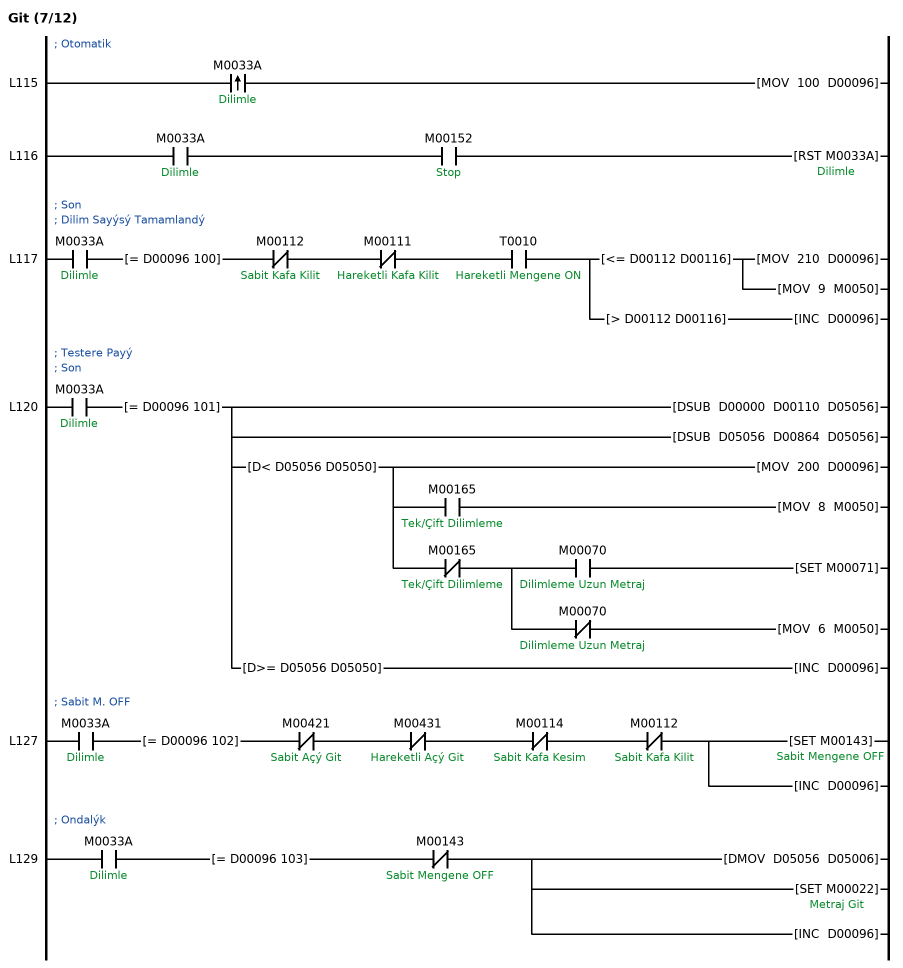
; L115
LOADP     M0033A	// Dilimle
MOV       100 D00096
// output comment: Otomatik
; L116
LOAD      M0033A	// Dilimle
AND       M00152	// Stop
RST       M0033A	// Dilimle
; L117
LOAD      M0033A	// Dilimle
AND=      D00096 100
AND NOT   M00112	// Sabit Kafa Kilit
AND NOT   M00111	// Hareketli Kafa Kilit
AND       T0010	// Hareketli Mengene ON
MPUSH
AND<=     D00112 D00116
MOV       210 D00096
MOV       9 M0050
MPOP
AND>      D00112 D00116
INC       D00096
// output comment: Son
// output comment: Dilim Sayýsý Tamamlandý
; L120
LOAD      M0033A	// Dilimle
AND=      D00096 101
DSUB      D00000 D00110 D05056
DSUB      D05056 D00864 D05056
MPUSH
ANDD<     D05056 D05050
MOV       200 D00096
MPUSH
AND       M00165	// Tek/Çift Dilimleme
MOV       8 M0050
MPOP
AND NOT   M00165	// Tek/Çift Dilimleme
MPUSH
AND       M00070	// Dilimleme Uzun Metraj
SET       M00071
MPOP
AND NOT   M00070	// Dilimleme Uzun Metraj
MOV       6 M0050
MPOP
ANDD>=    D05056 D05050
INC       D00096
// output comment: Testere Payý
// output comment: Son
; L127
LOAD      M0033A	// Dilimle
AND=      D00096 102
AND NOT   M00421	// Sabit Açý Git
AND NOT   M00431	// Hareketli Açý Git
AND NOT   M00114	// Sabit Kafa Kesim
AND NOT   M00112	// Sabit Kafa Kilit
SET       M00143	// Sabit Mengene OFF
INC       D00096
// output comment: Sabit M. OFF
; L129
LOAD      M0033A	// Dilimle
AND=      D00096 103
AND NOT   M00143	// Sabit Mengene OFF
DMOV      D05056 D05006
SET       M00022	// Metraj Git
INC       D00096
// output comment: Ondalýk

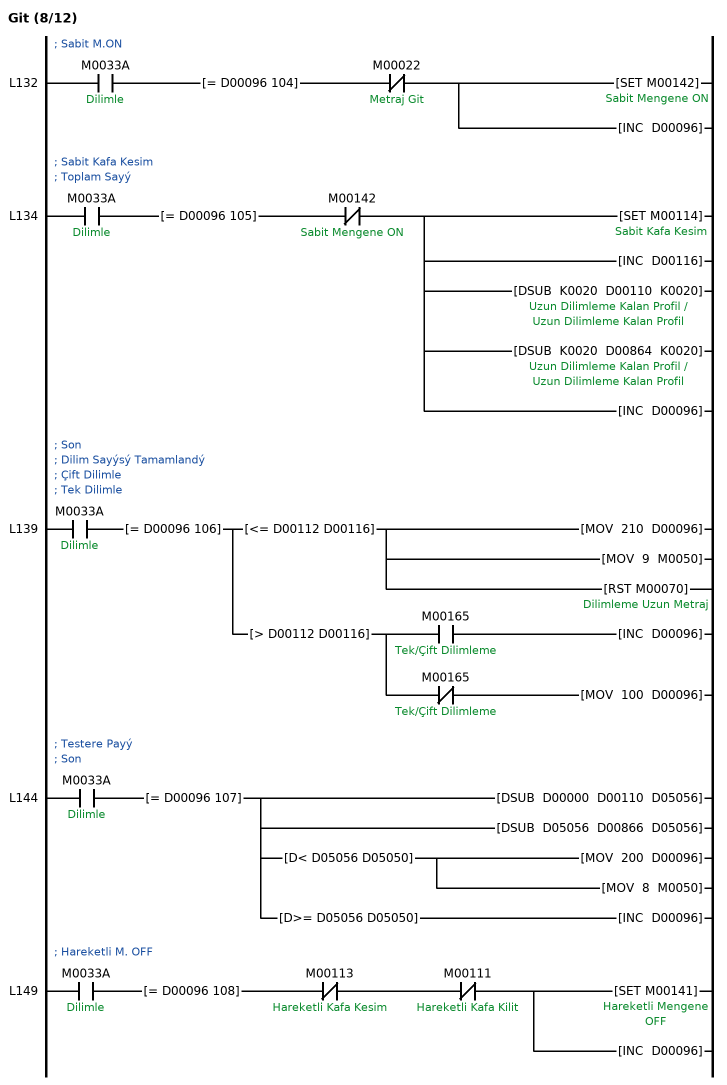
; L132
LOAD      M0033A	// Dilimle
AND=      D00096 104
AND NOT   M00022	// Metraj Git
SET       M00142	// Sabit Mengene ON
INC       D00096
// output comment: Sabit M.ON
; L134
LOAD      M0033A	// Dilimle
AND=      D00096 105
AND NOT   M00142	// Sabit Mengene ON
SET       M00114	// Sabit Kafa Kesim
INC       D00116
DSUB      K0020 D00110 K0020	// Uzun Dilimleme Kalan Profil / Uzun Dilimleme Kalan Profil
DSUB      K0020 D00864 K0020	// Uzun Dilimleme Kalan Profil / Uzun Dilimleme Kalan Profil
INC       D00096
// output comment: Sabit Kafa Kesim
// output comment: Toplam Sayý
; L139
LOAD      M0033A	// Dilimle
AND=      D00096 106
MPUSH
AND<=     D00112 D00116
MOV       210 D00096
MOV       9 M0050
RST       M00070	// Dilimleme Uzun Metraj
MPOP
AND>      D00112 D00116
MPUSH
AND       M00165	// Tek/Çift Dilimleme
INC       D00096
MPOP
AND NOT   M00165	// Tek/Çift Dilimleme
MOV       100 D00096
// output comment: Son
// output comment: Dilim Sayýsý Tamamlandý
// output comment: Çift Dilimle
// output comment: Tek Dilimle
; L144
LOAD      M0033A	// Dilimle
AND=      D00096 107
DSUB      D00000 D00110 D05056
DSUB      D05056 D00866 D05056
MPUSH
ANDD<     D05056 D05050
MOV       200 D00096
MOV       8 M0050
MPOP
ANDD>=    D05056 D05050
INC       D00096
// output comment: Testere Payý
// output comment: Son
; L149
LOAD      M0033A	// Dilimle
AND=      D00096 108
AND NOT   M00113	// Hareketli Kafa Kesim
AND NOT   M00111	// Hareketli Kafa Kilit
SET       M00141	// Hareketli Mengene OFF
INC       D00096
// output comment: Hareketli M. OFF

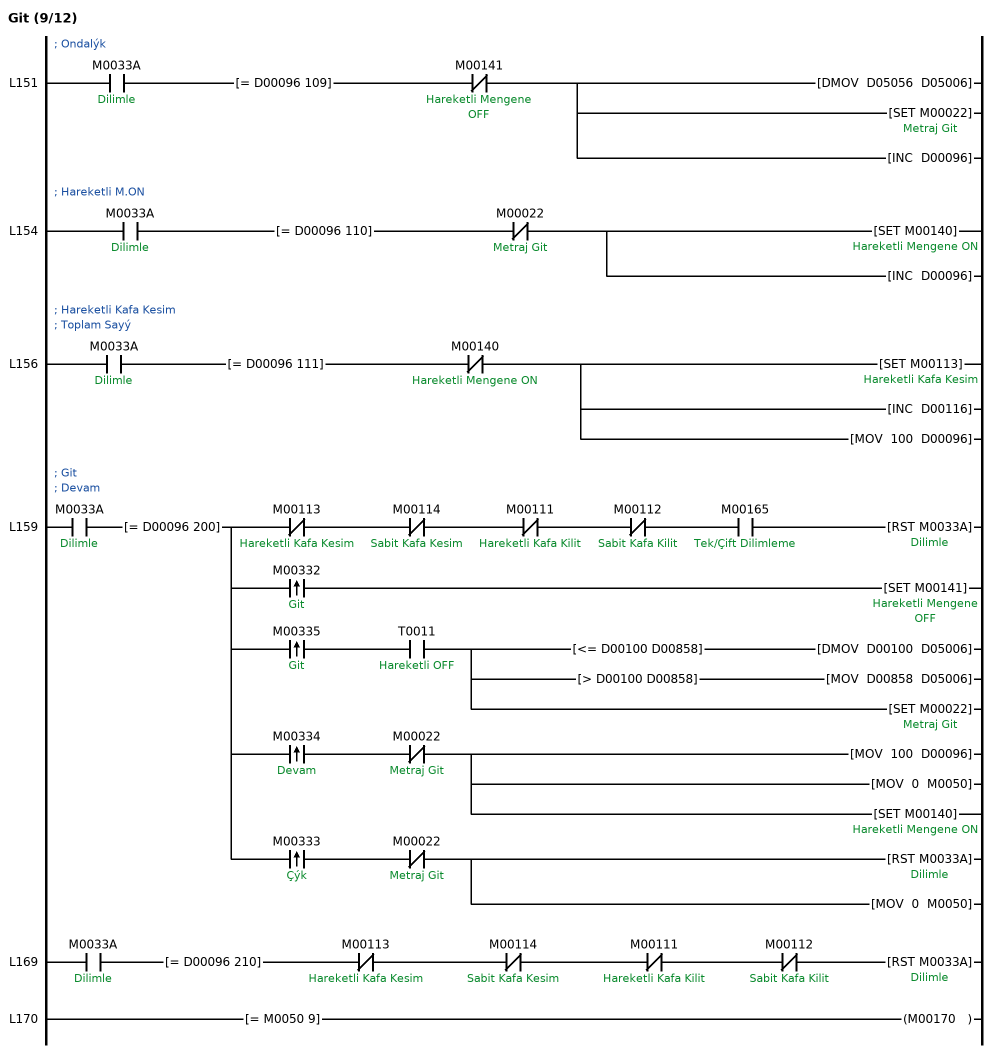
; L151
LOAD      M0033A	// Dilimle
AND=      D00096 109
AND NOT   M00141	// Hareketli Mengene OFF
DMOV      D05056 D05006
SET       M00022	// Metraj Git
INC       D00096
// output comment: Ondalýk
; L154
LOAD      M0033A	// Dilimle
AND=      D00096 110
AND NOT   M00022	// Metraj Git
SET       M00140	// Hareketli Mengene ON
INC       D00096
// output comment: Hareketli M.ON
; L156
LOAD      M0033A	// Dilimle
AND=      D00096 111
AND NOT   M00140	// Hareketli Mengene ON
SET       M00113	// Hareketli Kafa Kesim
INC       D00116
MOV       100 D00096
// output comment: Hareketli Kafa Kesim
// output comment: Toplam Sayý
; L159
LOAD      M0033A	// Dilimle
AND=      D00096 200
MPUSH
AND NOT   M00113	// Hareketli Kafa Kesim
AND NOT   M00114	// Sabit Kafa Kesim
AND NOT   M00111	// Hareketli Kafa Kilit
AND NOT   M00112	// Sabit Kafa Kilit
AND       M00165	// Tek/Çift Dilimleme
RST       M0033A	// Dilimle
MLOAD
ANDP      M00332	// Git
SET       M00141	// Hareketli Mengene OFF
MLOAD
ANDP      M00335	// Git
AND       T0011	// Hareketli OFF
MPUSH
AND<=     D00100 D00858
DMOV      D00100 D05006
MLOAD
AND>      D00100 D00858
MOV       D00858 D05006
MPOP
SET       M00022	// Metraj Git
MLOAD
ANDP      M00334	// Devam
AND NOT   M00022	// Metraj Git
MOV       100 D00096
MOV       0 M0050
SET       M00140	// Hareketli Mengene ON
MPOP
ANDP      M00333	// Çýk
AND NOT   M00022	// Metraj Git
RST       M0033A	// Dilimle
MOV       0 M0050
// output comment: Git
// output comment: Devam
; L169
LOAD      M0033A	// Dilimle
AND=      D00096 210
AND NOT   M00113	// Hareketli Kafa Kesim
AND NOT   M00114	// Sabit Kafa Kesim
AND NOT   M00111	// Hareketli Kafa Kilit
AND NOT   M00112	// Sabit Kafa Kilit
RST       M0033A	// Dilimle
; L170
LOAD=     M0050 9
OUT       M00170

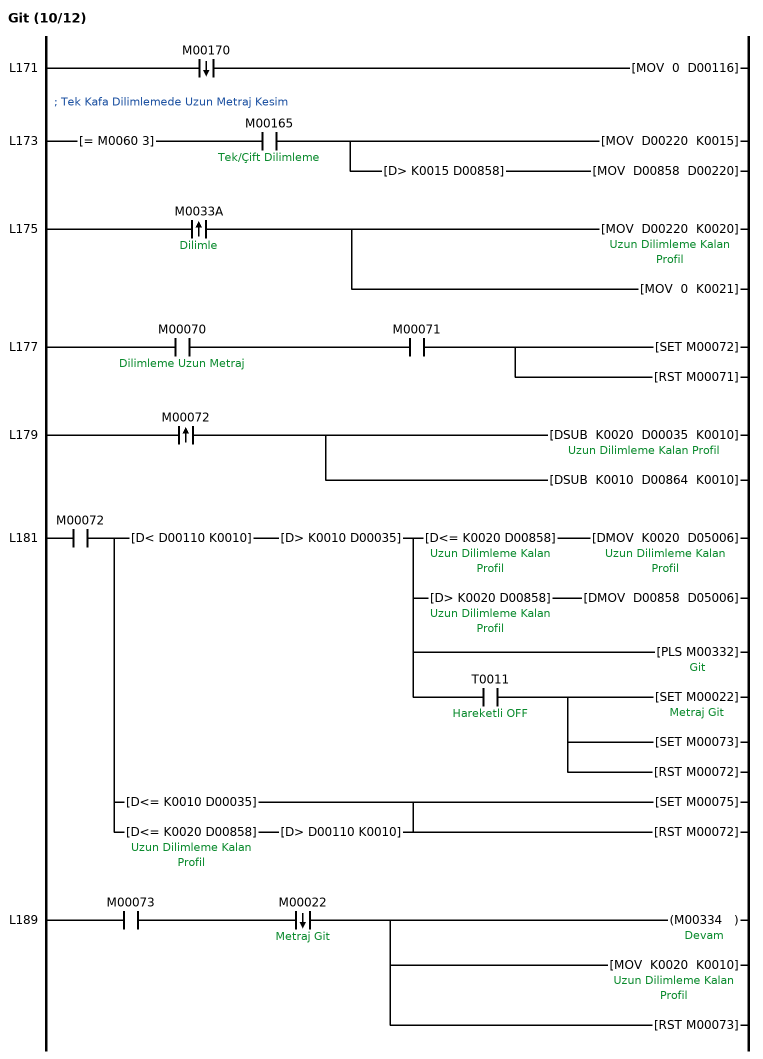
; L171
LOADN     M00170
MOV       0 D00116
// Tek Kafa Dilimlemede Uzun Metraj Kesim
; L173
LOAD=     M0060 3
AND       M00165	// Tek/Çift Dilimleme
MOV       D00220 K0015
ANDD>     K0015 D00858
MOV       D00858 D00220
; L175
LOADP     M0033A	// Dilimle
MOV       D00220 K0020	// Uzun Dilimleme Kalan Profil
MOV       0 K0021
; L177
LOAD      M00070	// Dilimleme Uzun Metraj
AND       M00071
SET       M00072
RST       M00071
; L179
LOADP     M00072
DSUB      K0020 D00035 K0010	// Uzun Dilimleme Kalan Profil
DSUB      K0010 D00864 K0010
; L181
LOAD      M00072
MPUSH
ANDD<     D00110 K0010
ANDD>     K0010 D00035
MPUSH
ANDD<=    K0020 D00858	// Uzun Dilimleme Kalan Profil
DMOV      K0020 D05006	// Uzun Dilimleme Kalan Profil
MLOAD
ANDD>     K0020 D00858	// Uzun Dilimleme Kalan Profil
DMOV      D00858 D05006
MPOP
OUTP      M00332	// Git
AND       T0011	// Hareketli OFF
SET       M00022	// Metraj Git
SET       M00073
RST       M00072
MPOP
LOADD<=   K0010 D00035
LOADD<=   K0020 D00858	// Uzun Dilimleme Kalan Profil
ANDD>     D00110 K0010
OR LOAD
AND LOAD
SET       M00075
RST       M00072
; L189
LOAD      M00073
ANDN      M00022	// Metraj Git
OUT       M00334	// Devam
MOV       K0020 K0010	// Uzun Dilimleme Kalan Profil
RST       M00073

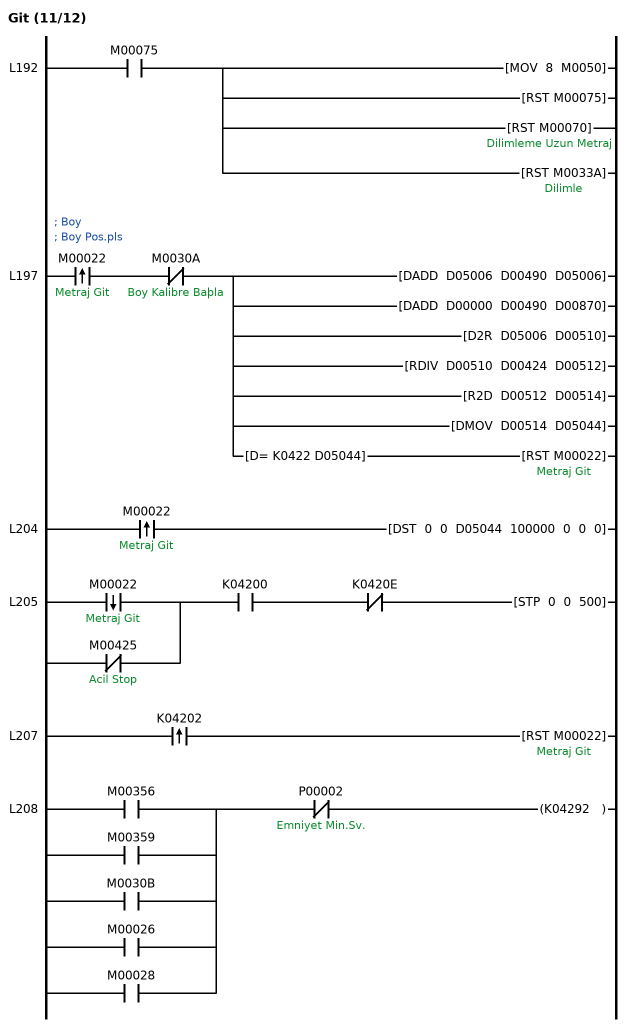
; L192
LOAD      M00075
MOV       8 M0050
RST       M00075
RST       M00070	// Dilimleme Uzun Metraj
RST       M0033A	// Dilimle
// Boy
; L197
LOADP     M00022	// Metraj Git
AND NOT   M0030A	// Boy Kalibre Baþla
DADD      D05006 D00490 D05006
DADD      D00000 D00490 D00870
D2R       D05006 D00510
RDIV      D00510 D00424 D00512
R2D       D00512 D00514
DMOV      D00514 D05044
ANDD=     K0422 D05044
RST       M00022	// Metraj Git
// output comment: Boy Pos.pls
; L204
LOADP     M00022	// Metraj Git
DST       0 0 D05044 100000 0 0 0
; L205
LOADN     M00022	// Metraj Git
OR NOT    M00425	// Acil Stop
AND       K04200
AND NOT   K0420E
STP       0 0 500
; L207
LOADP     K04202
RST       M00022	// Metraj Git
; L208
LOAD      M00356
OR        M00359
OR        M0030B
OR        M00026
OR        M00028
AND NOT   P00002	// Emniyet Min.Sv.
OUT       K04292

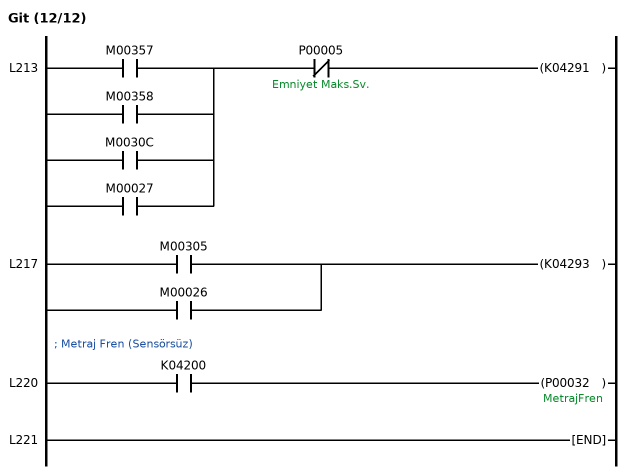
; L213
LOAD      M00357
OR        M00358
OR        M0030C
OR        M00027
AND NOT   P00005	// Emniyet Maks.Sv.
OUT       K04291
; L217
LOAD      M00305
OR        M00026
OUT       K04293
// Metraj Fren (Sensörsüz)
; L220
LOAD      K04200
OUT       P00032	// MetrajFren
; L221
END

PROGRAM Reçete (task: Scan Program)

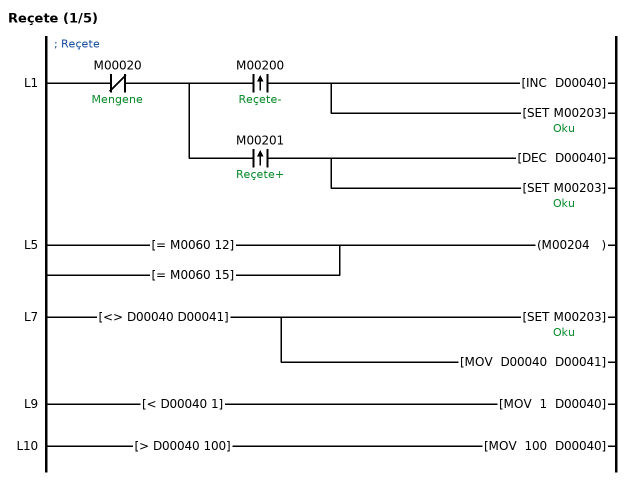
// Reçete
; L1
LOAD NOT  M00020	// Mengene
MPUSH
ANDP      M00200	// Reçete-
INC       D00040
SET       M00203	// Oku
MPOP
ANDP      M00201	// Reçete+
DEC       D00040
SET       M00203	// Oku
; L5
LOAD=     M0060 12
OR=       M0060 15
OUT       M00204
; L7
LOAD<>    D00040 D00041
SET       M00203	// Oku
MOV       D00040 D00041
; L9
LOAD<     D00040 1
MOV       1 D00040
; L10
LOAD>     D00040 100
MOV       100 D00040

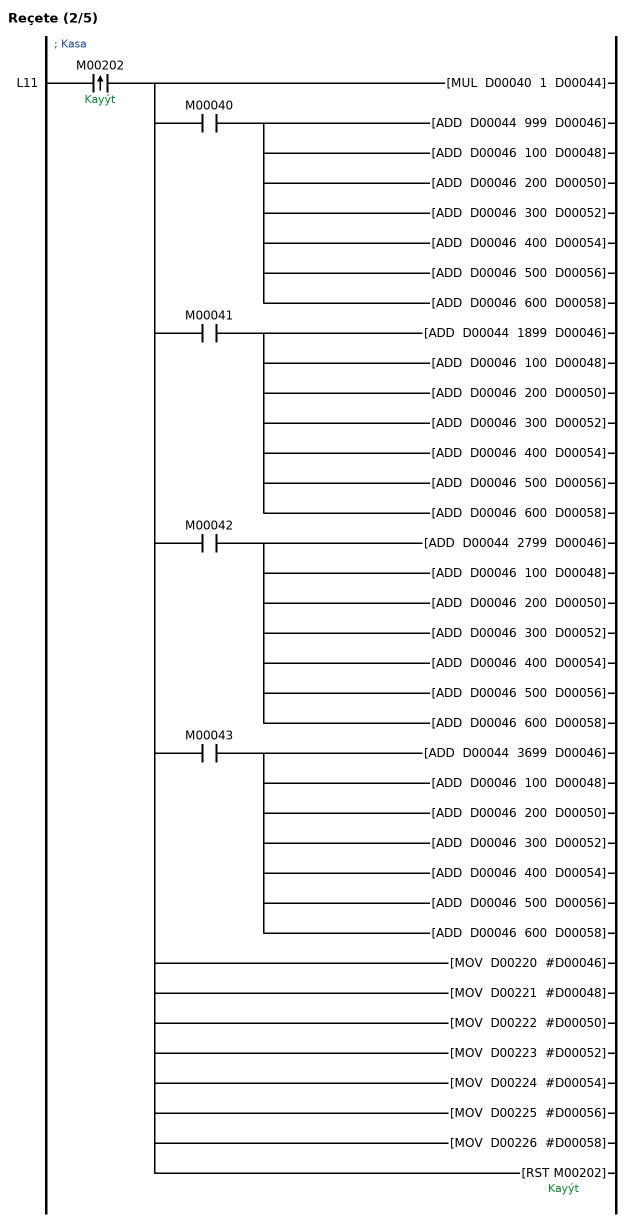
; L11
LOADP     M00202	// Kayýt
MUL       D00040 1 D00044
MPUSH
AND       M00040
ADD       D00044 999 D00046
ADD       D00046 100 D00048
ADD       D00046 200 D00050
ADD       D00046 300 D00052
ADD       D00046 400 D00054
ADD       D00046 500 D00056
ADD       D00046 600 D00058
MLOAD
AND       M00041
ADD       D00044 1899 D00046
ADD       D00046 100 D00048
ADD       D00046 200 D00050
ADD       D00046 300 D00052
ADD       D00046 400 D00054
ADD       D00046 500 D00056
ADD       D00046 600 D00058
MLOAD
AND       M00042
ADD       D00044 2799 D00046
ADD       D00046 100 D00048
ADD       D00046 200 D00050
ADD       D00046 300 D00052
ADD       D00046 400 D00054
ADD       D00046 500 D00056
ADD       D00046 600 D00058
MLOAD
AND       M00043
ADD       D00044 3699 D00046
ADD       D00046 100 D00048
ADD       D00046 200 D00050
ADD       D00046 300 D00052
ADD       D00046 400 D00054
ADD       D00046 500 D00056
ADD       D00046 600 D00058
MPOP
MOV       D00220 #D00046
MOV       D00221 #D00048
MOV       D00222 #D00050
MOV       D00223 #D00052
MOV       D00224 #D00054
MOV       D00225 #D00056
MOV       D00226 #D00058
RST       M00202	// Kayýt
// output comment: Kasa

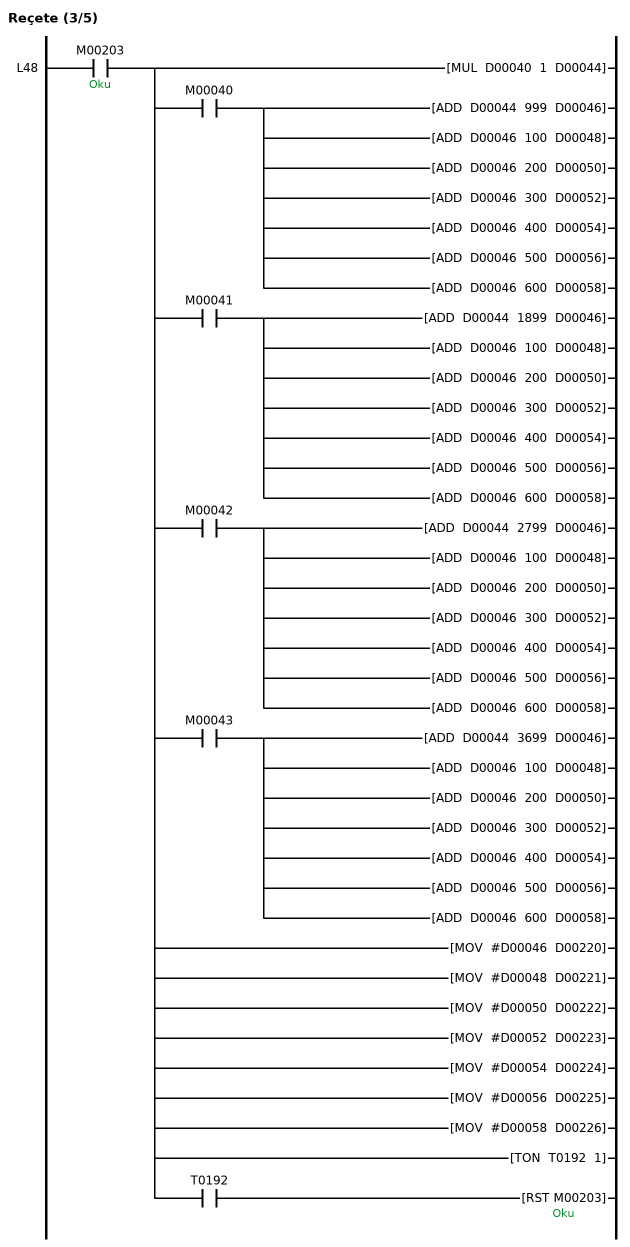
; L48
LOAD      M00203	// Oku
MUL       D00040 1 D00044
MPUSH
AND       M00040
ADD       D00044 999 D00046
ADD       D00046 100 D00048
ADD       D00046 200 D00050
ADD       D00046 300 D00052
ADD       D00046 400 D00054
ADD       D00046 500 D00056
ADD       D00046 600 D00058
MLOAD
AND       M00041
ADD       D00044 1899 D00046
ADD       D00046 100 D00048
ADD       D00046 200 D00050
ADD       D00046 300 D00052
ADD       D00046 400 D00054
ADD       D00046 500 D00056
ADD       D00046 600 D00058
MLOAD
AND       M00042
ADD       D00044 2799 D00046
ADD       D00046 100 D00048
ADD       D00046 200 D00050
ADD       D00046 300 D00052
ADD       D00046 400 D00054
ADD       D00046 500 D00056
ADD       D00046 600 D00058
MLOAD
AND       M00043
ADD       D00044 3699 D00046
ADD       D00046 100 D00048
ADD       D00046 200 D00050
ADD       D00046 300 D00052
ADD       D00046 400 D00054
ADD       D00046 500 D00056
ADD       D00046 600 D00058
MPOP
MOV       #D00046 D00220
MOV       #D00048 D00221
MOV       #D00050 D00222
MOV       #D00052 D00223
MOV       #D00054 D00224
MOV       #D00056 D00225
MOV       #D00058 D00226
TON       T0192 1
AND       T0192
RST       M00203	// Oku

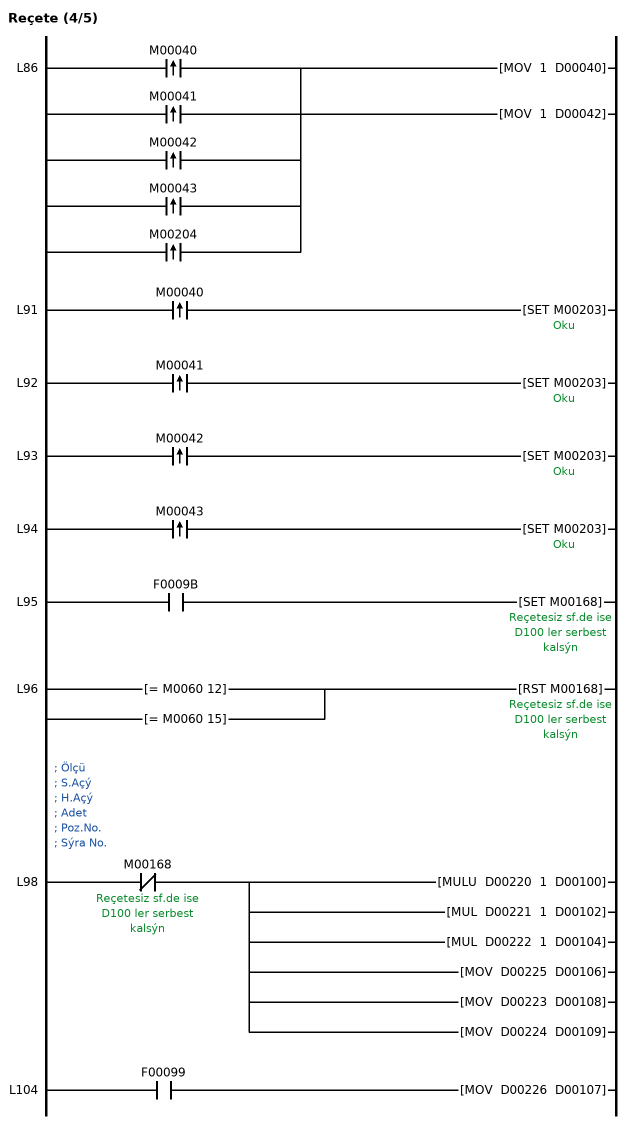
; L86
LOADP     M00040
ORP       M00041
ORP       M00042
ORP       M00043
ORP       M00204
MOV       1 D00040
MOV       1 D00042
; L91
LOADP     M00040
SET       M00203	// Oku
; L92
LOADP     M00041
SET       M00203	// Oku
; L93
LOADP     M00042
SET       M00203	// Oku
; L94
LOADP     M00043
SET       M00203	// Oku
; L95
LOAD      F0009B
SET       M00168	// Reçetesiz sf.de ise D100 ler serbest kalsýn
; L96
LOAD=     M0060 12
OR=       M0060 15
RST       M00168	// Reçetesiz sf.de ise D100 ler serbest kalsýn
; L98
LOAD NOT  M00168	// Reçetesiz sf.de ise D100 ler serbest kalsýn
MULU      D00220 1 D00100
MUL       D00221 1 D00102
MUL       D00222 1 D00104
MOV       D00225 D00106
MOV       D00223 D00108
MOV       D00224 D00109
// output comment: Ölçü
// output comment: S.Açý
// output comment: H.Açý
// output comment: Adet
// output comment: Poz.No.
// output comment: Sýra No.
; L104
LOAD      F00099
MOV       D00226 D00107

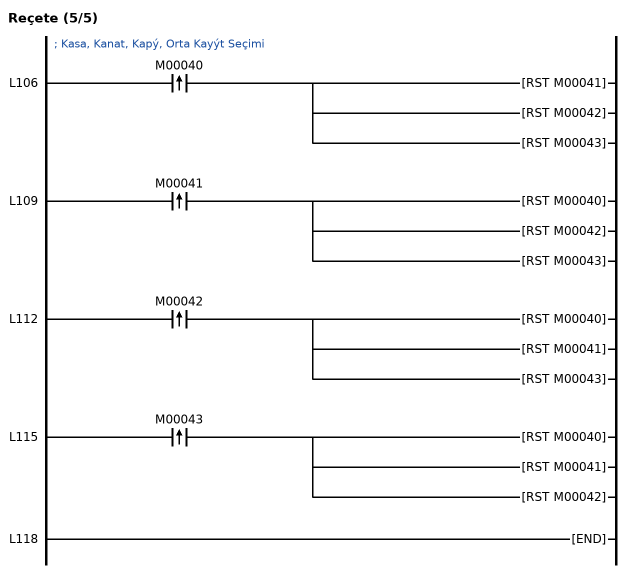
// Kasa, Kanat, Kapý, Orta Kayýt Seçimi
; L106
LOADP     M00040
RST       M00041
RST       M00042
RST       M00043
; L109
LOADP     M00041
RST       M00040
RST       M00042
RST       M00043
; L112
LOADP     M00042
RST       M00040
RST       M00041
RST       M00043
; L115
LOADP     M00043
RST       M00040
RST       M00041
RST       M00042
; L118
END

PROGRAM Sabitler (task: Scan Program)

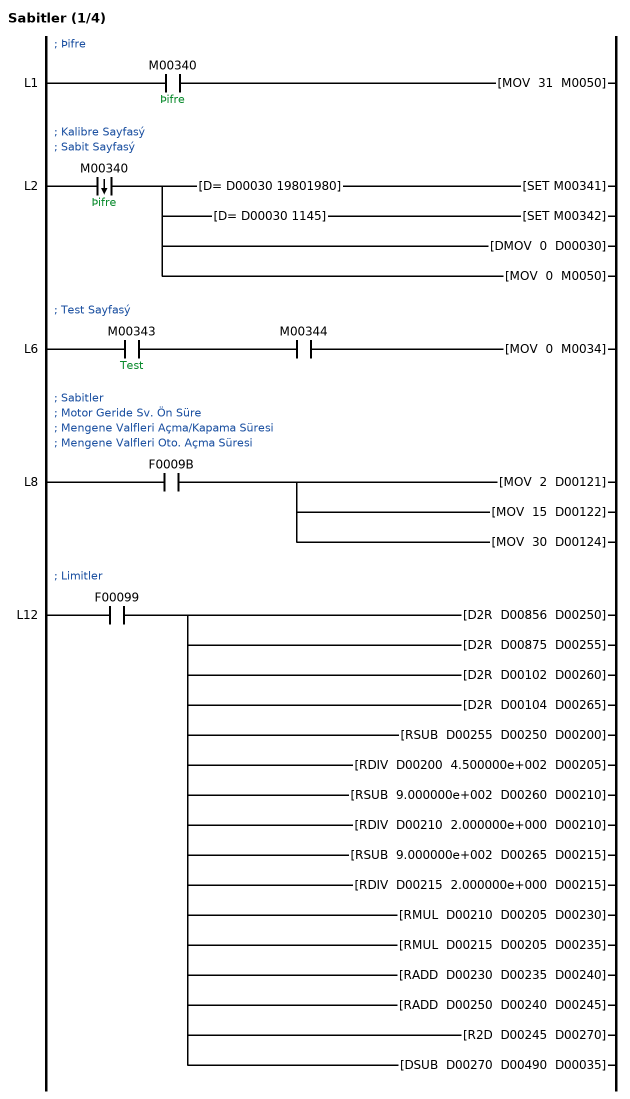
// Þifre
; L1
LOAD      M00340	// Þifre
MOV       31 M0050
; L2
LOADN     M00340	// Þifre
MPUSH
ANDD=     D00030 19801980
SET       M00341
MLOAD
ANDD=     D00030 1145
SET       M00342
MPOP
DMOV      0 D00030
MOV       0 M0050
// output comment: Kalibre Sayfasý
// output comment: Sabit Sayfasý
; L6
LOAD      M00343	// Test
AND       M00344
MOV       0 M0034
// output comment: Test Sayfasý
// Sabitler
; L8
LOAD      F0009B
MOV       2 D00121
MOV       15 D00122
MOV       30 D00124
// output comment: Motor Geride Sv. Ön Süre
// output comment: Mengene Valfleri Açma/Kapama Süresi
// output comment: Mengene Valfleri Oto. Açma Süresi
// Limitler
; L12
LOAD      F00099
D2R       D00856 D00250
D2R       D00875 D00255
D2R       D00102 D00260
D2R       D00104 D00265
RSUB      D00255 D00250 D00200
RDIV      D00200 4.500000e+002 D00205
RSUB      9.000000e+002 D00260 D00210
RDIV      D00210 2.000000e+000 D00210
RSUB      9.000000e+002 D00265 D00215
RDIV      D00215 2.000000e+000 D00215
RMUL      D00210 D00205 D00230
RMUL      D00215 D00205 D00235
RADD      D00230 D00235 D00240
RADD      D00250 D00240 D00245
R2D       D00245 D00270
DSUB      D00270 D00490 D00035

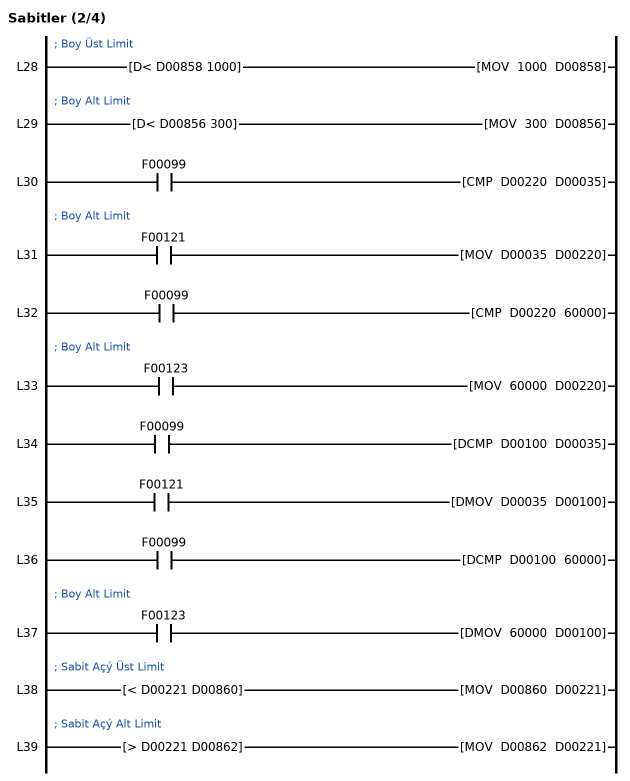
; L28
LOADD<    D00858 1000
MOV       1000 D00858
// output comment: Boy Üst Limit
; L29
LOADD<    D00856 300
MOV       300 D00856
// output comment: Boy Alt Limit
; L30
LOAD      F00099
CMP       D00220 D00035
; L31
LOAD      F00121
MOV       D00035 D00220
// output comment: Boy Alt Limit
; L32
LOAD      F00099
CMP       D00220 60000
; L33
LOAD      F00123
MOV       60000 D00220
// output comment: Boy Alt Limit
; L34
LOAD      F00099
DCMP      D00100 D00035
; L35
LOAD      F00121
DMOV      D00035 D00100
; L36
LOAD      F00099
DCMP      D00100 60000
; L37
LOAD      F00123
DMOV      60000 D00100
// output comment: Boy Alt Limit
; L38
LOAD<     D00221 D00860
MOV       D00860 D00221
// output comment: Sabit Açý Üst Limit
; L39
LOAD>     D00221 D00862
MOV       D00862 D00221
// output comment: Sabit Açý Alt Limit

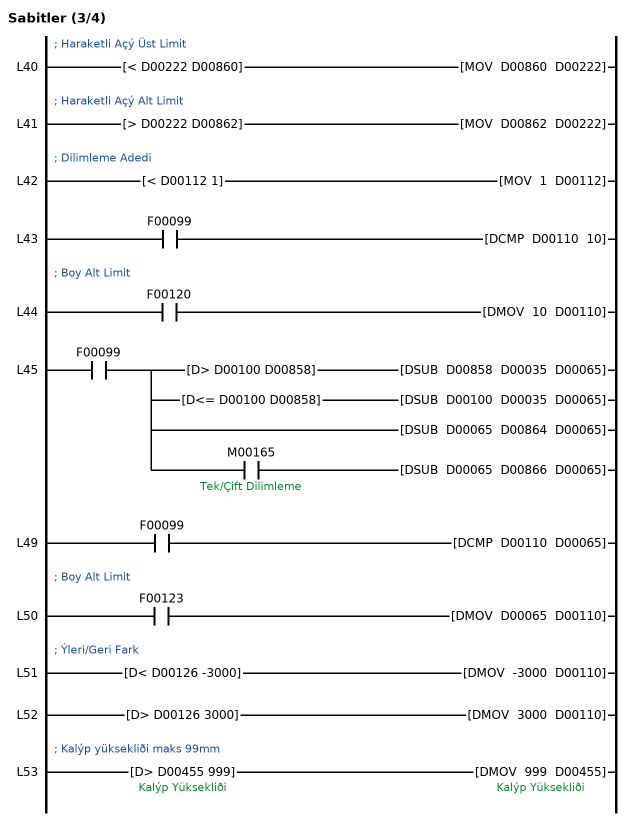
; L40
LOAD<     D00222 D00860
MOV       D00860 D00222
// output comment: Haraketli Açý Üst Limit
; L41
LOAD>     D00222 D00862
MOV       D00862 D00222
// output comment: Haraketli Açý Alt Limit
; L42
LOAD<     D00112 1
MOV       1 D00112
// output comment: Dilimleme Adedi
; L43
LOAD      F00099
DCMP      D00110 10
; L44
LOAD      F00120
DMOV      10 D00110
// output comment: Boy Alt Limit
; L45
LOAD      F00099
MPUSH
ANDD>     D00100 D00858
DSUB      D00858 D00035 D00065
MLOAD
ANDD<=    D00100 D00858
DSUB      D00100 D00035 D00065
MPOP
DSUB      D00065 D00864 D00065
AND       M00165	// Tek/Çift Dilimleme
DSUB      D00065 D00866 D00065
; L49
LOAD      F00099
DCMP      D00110 D00065
; L50
LOAD      F00123
DMOV      D00065 D00110
// output comment: Boy Alt Limit
; L51
LOADD<    D00126 -3000
DMOV      -3000 D00110
// output comment: Ýleri/Geri Fark
; L52
LOADD>    D00126 3000
DMOV      3000 D00110
; L53
LOADD>    D00455 999	// Kalýp Yüksekliði
DMOV      999 D00455	// Kalýp Yüksekliði
// output comment: Kalýp yüksekliði maks 99mm

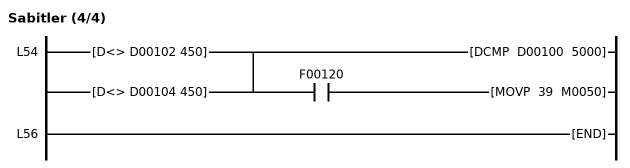
; L54
LOADD<>   D00102 450
ORD<>     D00104 450
DCMP      D00100 5000
AND       F00120
MOVP      39 M0050
; L56
END

PROGRAM Fuar modu (task: Scan Program)

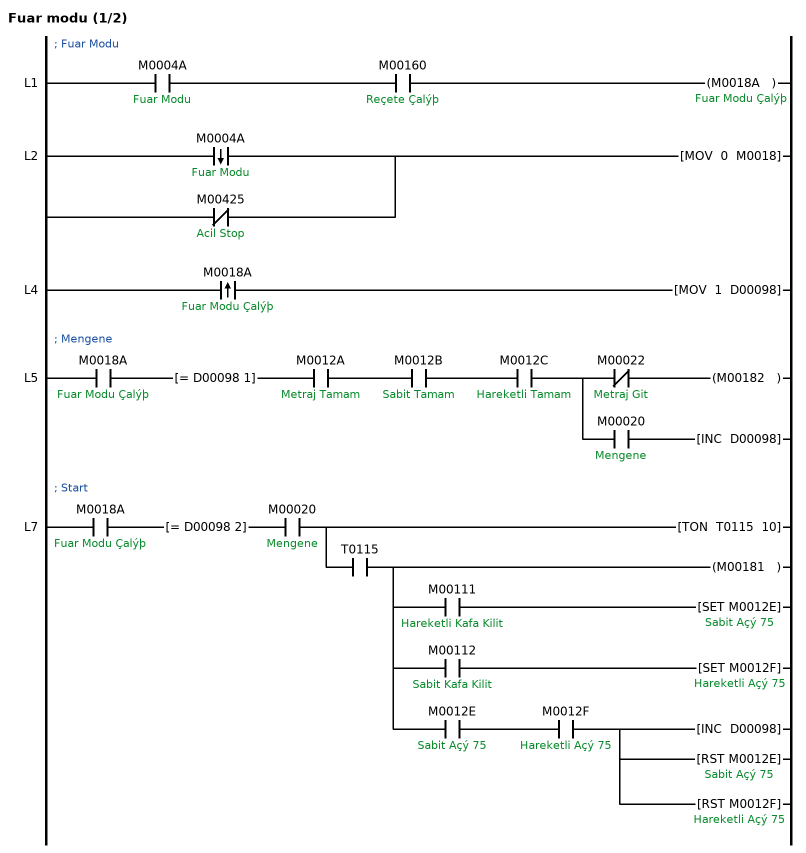
// Fuar Modu
; L1
LOAD      M0004A	// Fuar Modu
AND       M00160	// Reçete Çalýþ
OUT       M0018A	// Fuar Modu Çalýþ
; L2
LOADN     M0004A	// Fuar Modu
OR NOT    M00425	// Acil Stop
MOV       0 M0018
; L4
LOADP     M0018A	// Fuar Modu Çalýþ
MOV       1 D00098
; L5
LOAD      M0018A	// Fuar Modu Çalýþ
AND=      D00098 1
AND       M0012A	// Metraj Tamam
AND       M0012B	// Sabit Tamam
AND       M0012C	// Hareketli Tamam
MPUSH
AND NOT   M00022	// Metraj Git
OUT       M00182
MPOP
AND       M00020	// Mengene
INC       D00098
// output comment: Mengene
; L7
LOAD      M0018A	// Fuar Modu Çalýþ
AND=      D00098 2
AND       M00020	// Mengene
TON       T0115 10
AND       T0115
OUT       M00181
MPUSH
AND       M00111	// Hareketli Kafa Kilit
SET       M0012E	// Sabit Açý 75
MLOAD
AND       M00112	// Sabit Kafa Kilit
SET       M0012F	// Hareketli Açý 75
MPOP
AND       M0012E	// Sabit Açý 75
AND       M0012F	// Hareketli Açý 75
INC       D00098
RST       M0012E	// Sabit Açý 75
RST       M0012F	// Hareketli Açý 75
// output comment: Start

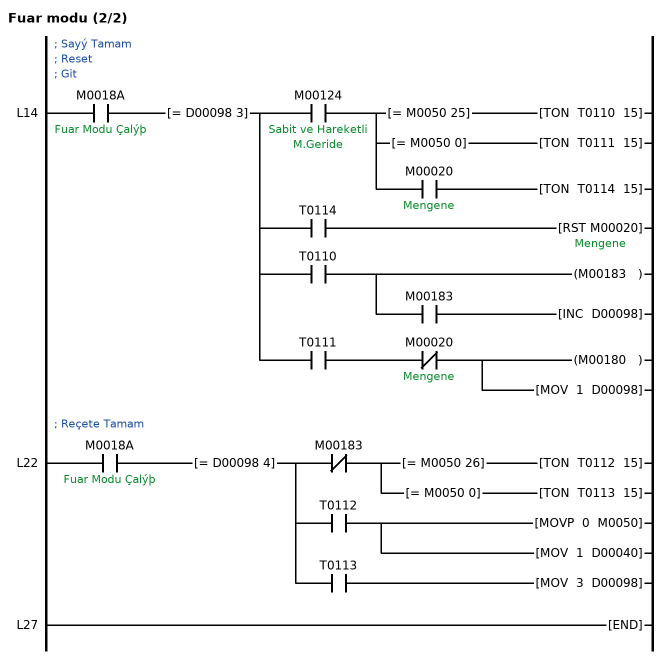
; L14
LOAD      M0018A	// Fuar Modu Çalýþ
AND=      D00098 3
MPUSH
AND       M00124	// Sabit ve Hareketli M.Geride
MPUSH
AND=      M0050 25
TON       T0110 15
MLOAD
AND=      M0050 0
TON       T0111 15
MPOP
AND       M00020	// Mengene
TON       T0114 15
MLOAD
AND       T0114
RST       M00020	// Mengene
MLOAD
AND       T0110
OUT       M00183
AND       M00183
INC       D00098
MPOP
AND       T0111
AND NOT   M00020	// Mengene
OUT       M00180
MOV       1 D00098
// output comment: Sayý Tamam
// output comment: Reset
// output comment: Git
; L22
LOAD      M0018A	// Fuar Modu Çalýþ
AND=      D00098 4
MPUSH
AND NOT   M00183
MPUSH
AND=      M0050 26
TON       T0112 15
MPOP
AND=      M0050 0
TON       T0113 15
MLOAD
AND       T0112
MOVP      0 M0050
MOV       1 D00040
MPOP
AND       T0113
MOV       3 D00098
// output comment: Reçete Tamam
; L27
END

PROGRAM Haberleþme (task: Scan Program)

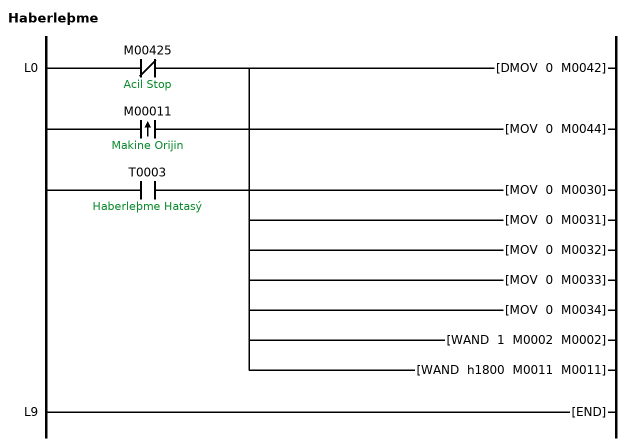
; L0
LOAD NOT  M00425	// Acil Stop
ORP       M00011	// Makine Orijin
OR        T0003	// Haberleþme Hatasý
DMOV      0 M0042
MOV       0 M0044
MOV       0 M0030
MOV       0 M0031
MOV       0 M0032
MOV       0 M0033
MOV       0 M0034
WAND      1 M0002 M0002
WAND      h1800 M0011 M0011
; L9
END

PROGRAM Kafalar (task: Scan Program)

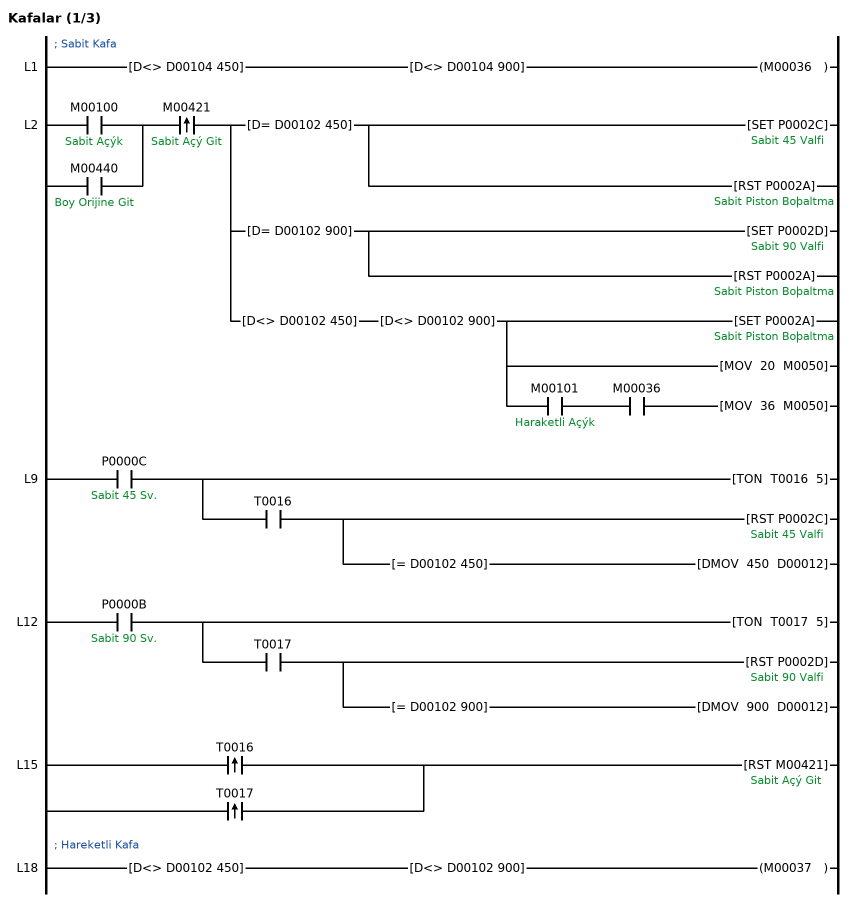
// Sabit Kafa
; L1
LOADD<>   D00104 450
ANDD<>    D00104 900
OUT       M00036
; L2
LOAD      M00100	// Sabit Açýk
OR        M00440	// Boy Orijine Git
ANDP      M00421	// Sabit Açý Git
MPUSH
ANDD=     D00102 450
SET       P0002C	// Sabit 45 Valfi
RST       P0002A	// Sabit Piston Boþaltma
MLOAD
ANDD=     D00102 900
SET       P0002D	// Sabit 90 Valfi
RST       P0002A	// Sabit Piston Boþaltma
MPOP
ANDD<>    D00102 450
ANDD<>    D00102 900
SET       P0002A	// Sabit Piston Boþaltma
MOV       20 M0050
AND       M00101	// Haraketli Açýk
AND       M00036
MOV       36 M0050
; L9
LOAD      P0000C	// Sabit 45 Sv.
TON       T0016 5
AND       T0016
RST       P0002C	// Sabit 45 Valfi
AND=      D00102 450
DMOV      450 D00012
; L12
LOAD      P0000B	// Sabit 90 Sv.
TON       T0017 5
AND       T0017
RST       P0002D	// Sabit 90 Valfi
AND=      D00102 900
DMOV      900 D00012
; L15
LOADP     T0016
ORP       T0017
RST       M00421	// Sabit Açý Git
// Hareketli Kafa
; L18
LOADD<>   D00102 450
ANDD<>    D00102 900
OUT       M00037

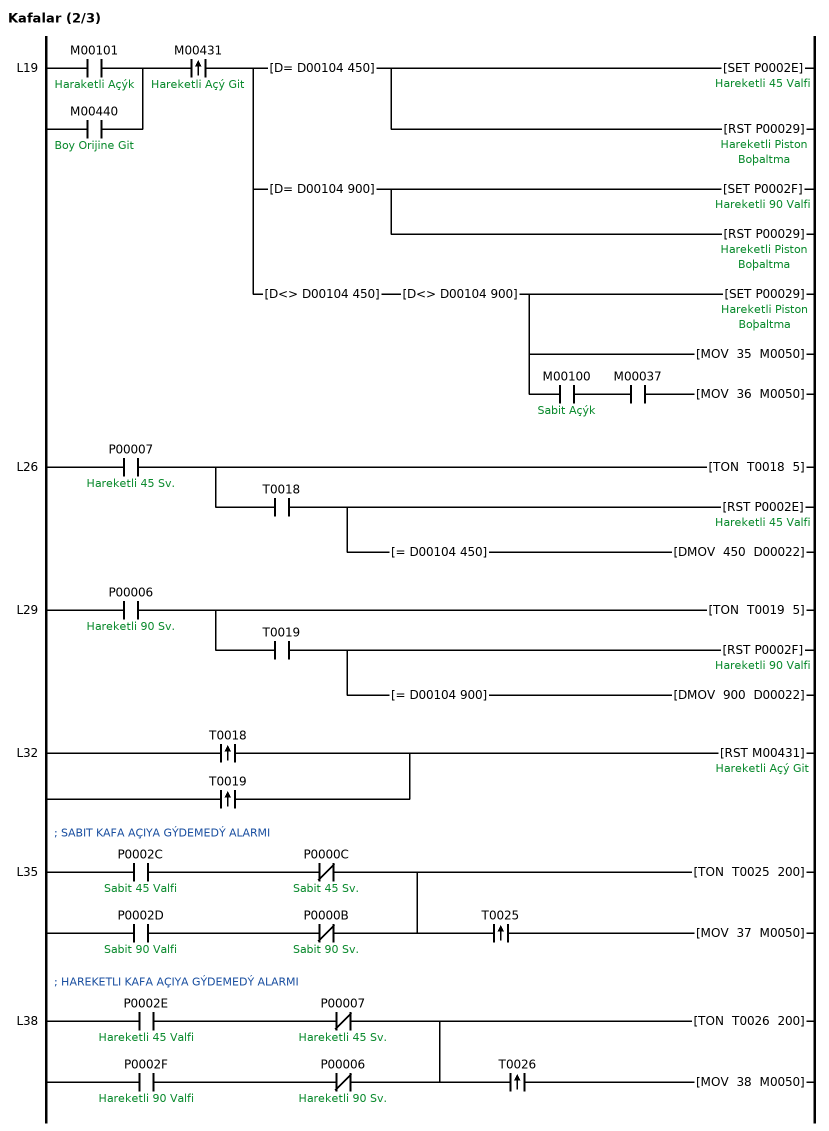
; L19
LOAD      M00101	// Haraketli Açýk
OR        M00440	// Boy Orijine Git
ANDP      M00431	// Hareketli Açý Git
MPUSH
ANDD=     D00104 450
SET       P0002E	// Hareketli 45 Valfi
RST       P00029	// Hareketli Piston Boþaltma
MLOAD
ANDD=     D00104 900
SET       P0002F	// Hareketli 90 Valfi
RST       P00029	// Hareketli Piston Boþaltma
MPOP
ANDD<>    D00104 450
ANDD<>    D00104 900
SET       P00029	// Hareketli Piston Boþaltma
MOV       35 M0050
AND       M00100	// Sabit Açýk
AND       M00037
MOV       36 M0050
; L26
LOAD      P00007	// Hareketli 45 Sv.
TON       T0018 5
AND       T0018
RST       P0002E	// Hareketli 45 Valfi
AND=      D00104 450
DMOV      450 D00022
; L29
LOAD      P00006	// Hareketli 90 Sv.
TON       T0019 5
AND       T0019
RST       P0002F	// Hareketli 90 Valfi
AND=      D00104 900
DMOV      900 D00022
; L32
LOADP     T0018
ORP       T0019
RST       M00431	// Hareketli Açý Git
// SABIT KAFA AÇIYA GÝDEMEDÝ ALARMI
; L35
LOAD      P0002C	// Sabit 45 Valfi
AND NOT   P0000C	// Sabit 45 Sv.
LOAD      P0002D	// Sabit 90 Valfi
AND NOT   P0000B	// Sabit 90 Sv.
OR LOAD
TON       T0025 200
ANDP      T0025
MOV       37 M0050
// HAREKETLI KAFA AÇIYA GÝDEMEDÝ ALARMI
; L38
LOAD      P0002E	// Hareketli 45 Valfi
AND NOT   P00007	// Hareketli 45 Sv.
LOAD      P0002F	// Hareketli 90 Valfi
AND NOT   P00006	// Hareketli 90 Sv.
OR LOAD
TON       T0026 200
ANDP      T0026
MOV       38 M0050

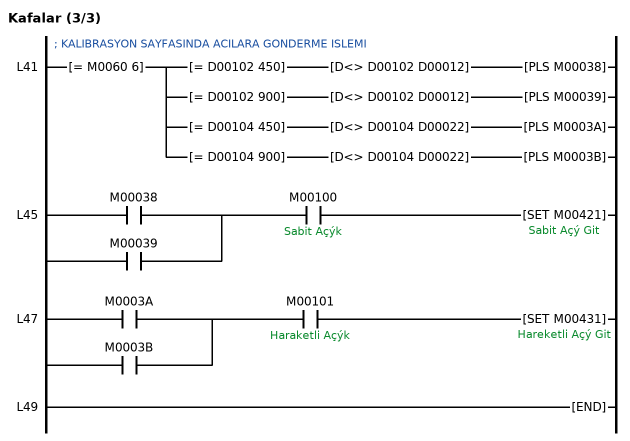
// KALIBRASYON SAYFASINDA ACILARA GONDERME ISLEMI
; L41
LOAD=     M0060 6
MPUSH
AND=      D00102 450
ANDD<>    D00102 D00012
OUTP      M00038
MLOAD
AND=      D00102 900
ANDD<>    D00102 D00012
OUTP      M00039
MLOAD
AND=      D00104 450
ANDD<>    D00104 D00022
OUTP      M0003A
MPOP
AND=      D00104 900
ANDD<>    D00104 D00022
OUTP      M0003B
; L45
LOAD      M00038
OR        M00039
AND       M00100	// Sabit Açýk
SET       M00421	// Sabit Açý Git
; L47
LOAD      M0003A
OR        M0003B
AND       M00101	// Haraketli Açýk
SET       M00431	// Hareketli Açý Git
; L49
END

PROGRAM Barkod yazýcý (task: Scan Program)

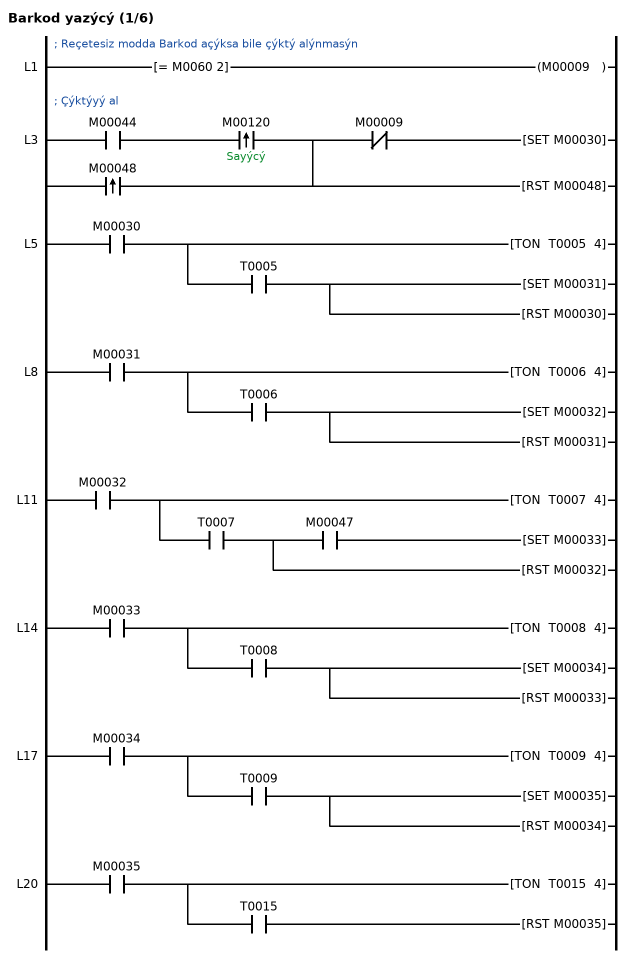
// Reçetesiz modda Barkod açýksa bile çýktý alýnmasýn
; L1
LOAD=     M0060 2
OUT       M00009
// Çýktýyý al
; L3
LOAD      M00044
ANDP      M00120	// Sayýcý
ORP       M00048
MPUSH
AND NOT   M00009
SET       M00030
MPOP
RST       M00048
; L5
LOAD      M00030
TON       T0005 4
AND       T0005
SET       M00031
RST       M00030
; L8
LOAD      M00031
TON       T0006 4
AND       T0006
SET       M00032
RST       M00031
; L11
LOAD      M00032
TON       T0007 4
AND       T0007
MPUSH
AND       M00047
SET       M00033
MPOP
RST       M00032
; L14
LOAD      M00033
TON       T0008 4
AND       T0008
SET       M00034
RST       M00033
; L17
LOAD      M00034
TON       T0009 4
AND       T0009
SET       M00035
RST       M00034
; L20
LOAD      M00035
TON       T0015 4
AND       T0015
RST       M00035

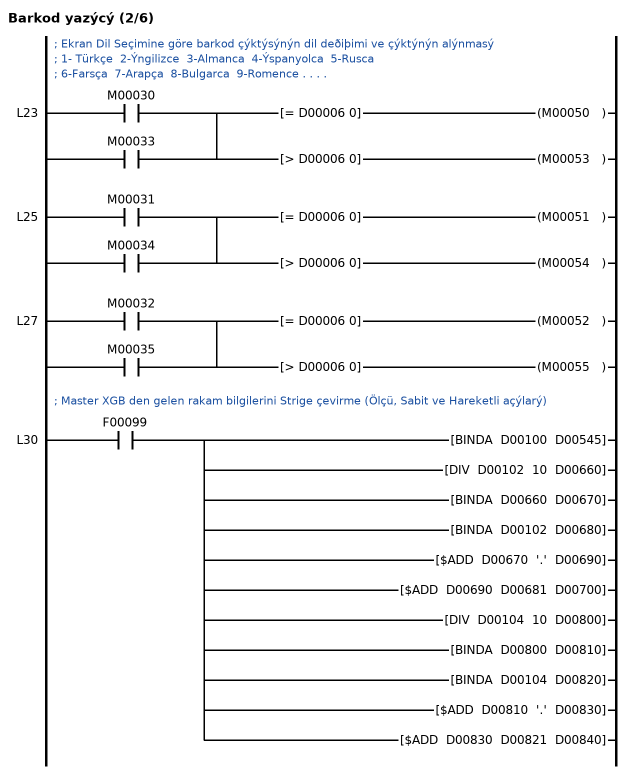
// Ekran Dil Seçimine göre barkod çýktýsýnýn dil deðiþimi ve çýktýnýn alýnmasý
// 1- Türkçe  2-Ýngilizce  3-Almanca  4-Ýspanyolca  5-Rusca
// 6-Farsça  7-Arapça  8-Bulgarca  9-Romence . . . .
; L23
LOAD      M00030
OR        M00033
MPUSH
AND=      D00006 0
OUT       M00050
MPOP
AND>      D00006 0
OUT       M00053
; L25
LOAD      M00031
OR        M00034
MPUSH
AND=      D00006 0
OUT       M00051
MPOP
AND>      D00006 0
OUT       M00054
; L27
LOAD      M00032
OR        M00035
MPUSH
AND=      D00006 0
OUT       M00052
MPOP
AND>      D00006 0
OUT       M00055
// Master XGB den gelen rakam bilgilerini Strige çevirme (Ölçü, Sabit ve Hareketli açýlarý)
; L30
LOAD      F00099
BINDA     D00100 D00545
DIV       D00102 10 D00660
BINDA     D00660 D00670
BINDA     D00102 D00680
$ADD      D00670 '.' D00690
$ADD      D00690 D00681 D00700
DIV       D00104 10 D00800
BINDA     D00800 D00810
BINDA     D00104 D00820
$ADD      D00810 '.' D00830
$ADD      D00830 D00821 D00840

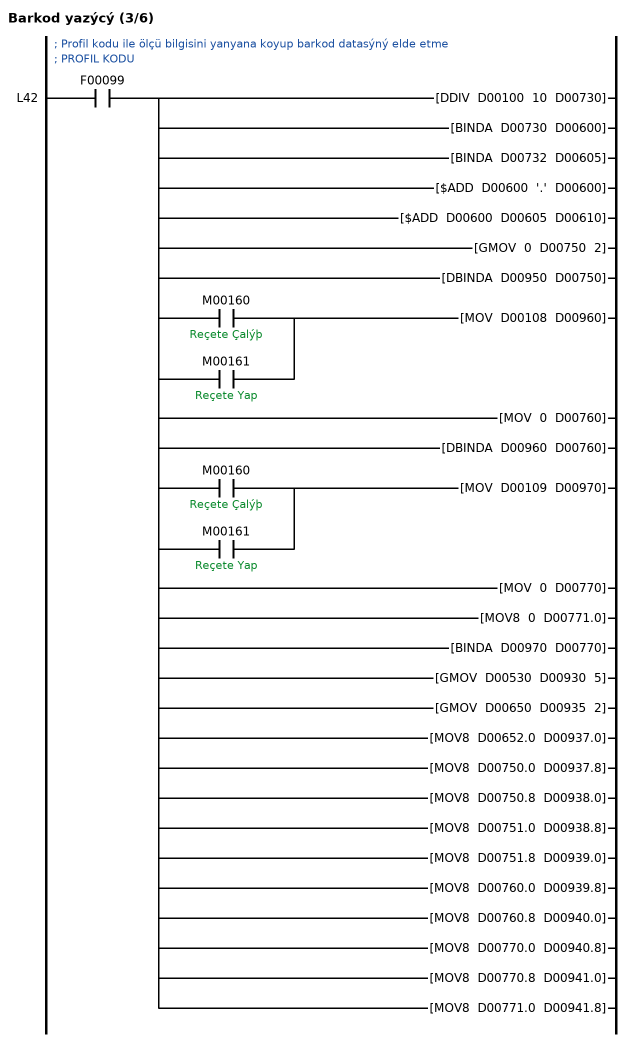
// Profil kodu ile ölçü bilgisini yanyana koyup barkod datasýný elde etme
; L42
LOAD      F00099
DDIV      D00100 10 D00730
BINDA     D00730 D00600
BINDA     D00732 D00605
$ADD      D00600 '.' D00600
$ADD      D00600 D00605 D00610
GMOV      0 D00750 2
DBINDA    D00950 D00750
MPUSH
LOAD      M00160	// Reçete Çalýþ
OR        M00161	// Reçete Yap
AND LOAD
MOV       D00108 D00960
MLOAD
MOV       0 D00760
DBINDA    D00960 D00760
LOAD      M00160	// Reçete Çalýþ
OR        M00161	// Reçete Yap
AND LOAD
MOV       D00109 D00970
MPOP
MOV       0 D00770
MOV8      0 D00771.0
BINDA     D00970 D00770
GMOV      D00530 D00930 5
GMOV      D00650 D00935 2
MOV8      D00652.0 D00937.0
MOV8      D00750.0 D00937.8
MOV8      D00750.8 D00938.0
MOV8      D00751.0 D00938.8
MOV8      D00751.8 D00939.0
MOV8      D00760.0 D00939.8
MOV8      D00760.8 D00940.0
MOV8      D00770.0 D00940.8
MOV8      D00770.8 D00941.0
MOV8      D00771.0 D00941.8
// output comment: PROFIL KODU

